(* IEC 61131-3 sources: agent_plc/, 3 files *)

(* ---- generated_traffic_light.st ---- *)
FUNCTION_BLOCK TrafficLightControl
VAR_INPUT
    manual_mode : BOOL;    (* Manual mode input *)
    emergency : BOOL;      (* Emergency button input *)
END_VAR

VAR_OUTPUT
    red_light : BOOL;      (* Red light output *)
    yellow_light : BOOL;   (* Yellow light output *)
    green_light : BOOL;    (* Green light output *)
END_VAR

VAR
    timer : TON;           (* Timer for state transitions *)
    state : INT := 0;      (* Current state: 0=Red, 1=Green, 2=Yellow *)
    timer_duration : TIME; (* Duration for the current state *)
    yellow_flash_state : BOOL := FALSE; (* Internal state for yellow light flashing *)
END_VAR

(* Main logic *)
IF manual_mode THEN
    (* Manual mode: Turn off all lights *)
    red_light := FALSE;
    yellow_light := FALSE;
    green_light := FALSE;
ELSIF emergency THEN
    (* Emergency mode: Yellow light flashes *)
    timer(IN := TRUE, PT := T#500ms); (* Flashing interval: 500ms *)
    IF timer.Q THEN
        yellow_flash_state := NOT yellow_flash_state; (* Toggle yellow light state *)
        timer(IN := FALSE); (* Reset timer *)
    END_IF;
    red_light := FALSE;
    yellow_light := yellow_flash_state;
    green_light := FALSE;
ELSE
    (* Normal mode: Traffic light sequence *)
    CASE state OF
        0: (* Red light state *)
            red_light := TRUE;
            yellow_light := FALSE;
            green_light := FALSE;
            timer_duration := T#30s; (* Red light duration *)
        1: (* Green light state *)
            red_light := FALSE;
            yellow_light := FALSE;
            green_light := TRUE;
            timer_duration := T#25s; (* Green light duration *)
        2: (* Yellow light state *)
            red_light := FALSE;
            yellow_light := TRUE;
            green_light := FALSE;
            timer_duration := T#5s; (* Yellow light duration *)
    END_CASE;

    (* Timer logic for state transitions *)
    timer(IN := TRUE, PT := timer_duration);
    IF timer.Q THEN
        timer(IN := FALSE); (* Reset timer *)
        state := (state + 1) MOD 3; (* Cycle through states: 0 -> 1 -> 2 -> 0 *)
    END_IF;
END_IF;

END_FUNCTION_BLOCK

(* ---- generated_traffic_light_complete.st ---- *)
FUNCTION_BLOCK TrafficLightControl
VAR_INPUT
    manual_mode : BOOL;    (* Manual mode input *)
    emergency : BOOL;      (* Emergency button input *)
END_VAR

VAR_OUTPUT
    red_light : BOOL;      (* Red light output *)
    yellow_light : BOOL;   (* Yellow light output *)
    green_light : BOOL;    (* Green light output *)
END_VAR

VAR
    timer : TON;           (* Timer for state transitions *)
    state : INT := 0;      (* Current state: 0=Red, 1=Green, 2=Yellow *)
    timer_duration : TIME; (* Duration for the current state *)
    yellow_flash_state : BOOL := FALSE; (* Internal state for yellow light flashing *)
END_VAR

(* Main logic *)
IF manual_mode THEN
    (* Manual mode: Turn off all lights *)
    red_light := FALSE;
    yellow_light := FALSE;
    green_light := FALSE;
ELSIF emergency THEN
    (* Emergency mode: Yellow light flashes *)
    timer(IN := TRUE, PT := T#500ms); (* Flashing interval: 500ms *)
    IF timer.Q THEN
        yellow_flash_state := NOT yellow_flash_state; (* Toggle yellow light state *)
        timer(IN := FALSE); (* Reset timer *)
    END_IF;
    red_light := FALSE;
    yellow_light := yellow_flash_state;
    green_light := FALSE;
ELSE
    (* Normal mode: Traffic light sequence *)
    CASE state OF
        0: (* Red light state *)
            red_light := TRUE;
            yellow_light := FALSE;
            green_light := FALSE;
            timer_duration := T#30s; (* Red light duration *)
        1: (* Green light state *)
            red_light := FALSE;
            yellow_light := FALSE;
            green_light := TRUE;
            timer_duration := T#25s; (* Green light duration *)
        2: (* Yellow light state *)
            red_light := FALSE;
            yellow_light := TRUE;
            green_light := FALSE;
            timer_duration := T#5s; (* Yellow light duration *)
    END_CASE;

    (* Timer logic for state transitions *)
    timer(IN := TRUE, PT := timer_duration);
    IF timer.Q THEN
        timer(IN := FALSE); (* Reset timer *)
        state := (state + 1) MOD 3; (* Cycle through states: 0 -> 1 -> 2 -> 0 *)
    END_IF;
END_IF;

END_FUNCTION_BLOCK

PROGRAM TrafficLight
VAR
    (* Input variables *)
    manual_mode : BOOL := FALSE;
    emergency : BOOL := FALSE;

    (* Output variables *)
    red_light : BOOL;
    yellow_light : BOOL;
    green_light : BOOL;

    (* Function block instance *)
    fb_traffic : TrafficLightControl;
END_VAR

(* Call function block *)
fb_traffic(
    manual_mode := manual_mode,
    emergency := emergency,
    red_light => red_light,
    yellow_light => yellow_light,
    green_light => green_light
);

END_PROGRAM

CONFIGURATION Config0
  RESOURCE Res0 ON PLC
    TASK Main(INTERVAL := T#100ms, PRIORITY := 0);
    PROGRAM Inst0 WITH Main : TrafficLight;
  END_RESOURCE
END_CONFIGURATION

(* ---- openplc_temp_simple.st ---- *)
PROGRAM TemperatureControl
VAR
    (* 输入变量 *)
    temperature : INT;      (* 温度传感器值 (0.01度精度) *)
    humidity : INT;         (* 湿度传感器值 (0.01%精度) *)
    manual_mode : BOOL;     (* 手动模式开关 *)

    (* 输出变量 *)
    heater : BOOL;          (* 加热器控制 *)
    cooler : BOOL;          (* 冷却器控制 *)
    fan : BOOL;             (* 排风扇控制 *)
    alarm : BOOL;           (* 报警指示 *)

    (* 内部变量 *)
    temp_real : REAL;       (* 实际温度值（浮点） *)
    hum_real : REAL;        (* 实际湿度值（浮点） *)
END_VAR

(* 转换输入为实数 *)
temp_real := INT_TO_REAL(temperature) / 100.0;
hum_real := INT_TO_REAL(humidity) / 100.0;

(* 手动模式检查 *)
IF manual_mode THEN
    (* 手动模式：关闭所有自动控制 *)
    heater := FALSE;
    cooler := FALSE;
    fan := FALSE;
    alarm := FALSE;
ELSE
    (* 自动模式 - 温度控制 *)
    IF temp_real < 18.0 THEN
        heater := TRUE;
        cooler := FALSE;
    ELSIF temp_real > 26.0 THEN
        cooler := TRUE;
        heater := FALSE;
    ELSE
        heater := FALSE;
        cooler := FALSE;
    END_IF;

    (* 湿度控制 *)
    IF hum_real > 70.0 THEN
        fan := TRUE;
    ELSE
        fan := FALSE;
    END_IF;

    (* 异常温度报警 *)
    IF (temp_real < 5.0) OR (temp_real > 40.0) THEN
        alarm := TRUE;
    ELSE
        alarm := FALSE;
    END_IF;
END_IF;

END_PROGRAM

CONFIGURATION Config0
  RESOURCE Res0 ON PLC
    TASK Main(INTERVAL := T#50ms, PRIORITY := 0);
    PROGRAM Inst0 WITH Main : TemperatureControl;
  END_RESOURCE
END_CONFIGURATION
